# EPICS autosave request: simDetectorApp/Db/simDetector_settings.req
$(P)$(R)GainX
$(P)$(R)GainY
$(P)$(R)GainRed
$(P)$(R)GainGreen
$(P)$(R)GainBlue
$(P)$(R)SimMode
$(P)$(R)PeakStartX
$(P)$(R)PeakStartY
$(P)$(R)PeakNumX
$(P)$(R)PeakNumY
$(P)$(R)PeakStepX
$(P)$(R)PeakStepY
$(P)$(R)PeakWidthX
$(P)$(R)PeakWidthY
$(P)$(R)PeakVariation
$(P)$(R)Noise
$(P)$(R)Offset
$(P)$(R)XSineOperation
$(P)$(R)XSine1Amplitude
$(P)$(R)XSine1Frequency
$(P)$(R)XSine1Phase
$(P)$(R)XSine2Amplitude
$(P)$(R)XSine2Frequency
$(P)$(R)XSine2Phase
$(P)$(R)YSineOperation
$(P)$(R)YSine1Amplitude
$(P)$(R)YSine1Frequency
$(P)$(R)YSine1Phase
$(P)$(R)YSine2Amplitude
$(P)$(R)YSine2Frequency
$(P)$(R)YSine2Phase
file "ADBase_settings.req", P=$(P), R=$(R)
